SUBAPPLICATION Uebung_217b_ALR (* Standard IEC 61131-3 ALI_FB_CTD (Adapter Version, LINT) mit Terminal-Ausgabe (PHYSA_LREAL) *)
  (* Standard: 61131-3; Description: Copyright (c) 2026 Meisterschulen am Ostbahnhof This program and the accompanying materials are made available under the terms of the Eclipse Public License 2.0 which is available at https://www.eclipse.org/legal/epl-2.0/ SPDX-License-Identifier: EPL-2.0 *)
  (* Version 1.2, 2026-05-13, Franz Höpfinger, Meisterschulen am Ostbahnhof, Added ALI_LINT_TO_LI init block connected to PV *)
  (* Version 1.1, 2026-04-21, Franz Höpfinger, Meisterschulen am Ostbahnhof, Added terminal output for counter value (PHYS) *)
  (* Version 1.0, 2026-04-21, Franz Höpfinger, Meisterschulen am Ostbahnhof, initial API and implementation (Adapter version) *)
  PACKAGE Uebungen;
  IMPORT Uebungen::const::UT::DefaultPool_Numeric::OutputNumber_N3_N;
  IMPORT logiBUS::io::DI::logiBUS_DI::Input_I1;
  IMPORT logiBUS::io::DI::logiBUS_DI::Input_I2;
  IMPORT logiBUS::io::DQ::logiBUS_DO::Output_Q1;
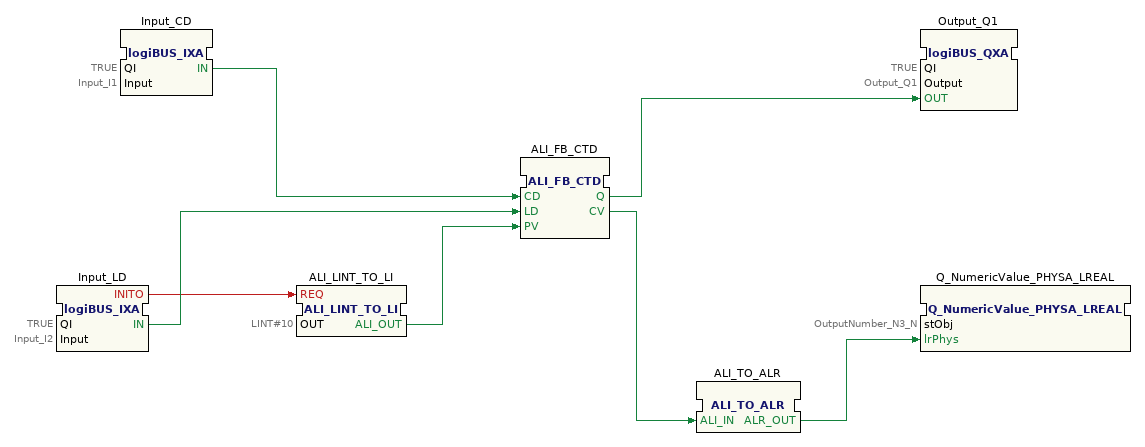
  (* hier sind negative Werte möglich ! *)
  (* hier gegebenenfalls einen AX_D_FF einbauen, damit die Events reduziert werden. *)
  FBS
    ALI_FB_CTD : adapter::iec61131::counters::ALI_FB_CTD;
    ALI_LINT_TO_LI : adapter::conversion::unidirectional::ALI_LINT_TO_LI(OUT := LINT#10);
    Input_CD : logiBUS::io::DI::logiBUS_IXA(QI := TRUE, Input := Input_I1);
    Input_LD : logiBUS::io::DI::logiBUS_IXA(QI := TRUE, Input := Input_I2);
    Output_Q1 : logiBUS::io::DQ::logiBUS_QXA(QI := TRUE, Output := Output_Q1);
    ALI_TO_ALR : adapter::conversion::unidirectional::ALI_TO_ALR;
    Q_NumericValue_PHYSA_LREAL : isobus::UT::Q::Q_NumericValue_PHYSA_LREAL(stObj := OutputNumber_N3_N);
  END_FBS
  EVENT_CONNECTIONS
    Input_LD.INITO TO ALI_LINT_TO_LI.REQ;
  END_CONNECTIONS
  ADAPTER_CONNECTIONS
    Input_CD.IN TO ALI_FB_CTD.CD;
    Input_LD.IN TO ALI_FB_CTD.LD;
    ALI_FB_CTD.Q TO Output_Q1.OUT;
    ALI_FB_CTD.CV TO ALI_TO_ALR.ALI_IN;
    ALI_TO_ALR.ALR_OUT TO Q_NumericValue_PHYSA_LREAL.lrPhys;
    ALI_LINT_TO_LI.ALI_OUT TO ALI_FB_CTD.PV;
  END_CONNECTIONS
END_SUBAPPLICATION
